(* IEC 61131-3 sources: DemoPumpStation/PumpStation/adapters/Codecs, 3 files *)

(* ---- modbus_base_codec.st ---- *)
class ModbusBaseCodec

var protected
        offset : udint := 0;
        segment : Modbus.IModbusSegmentAccess;
end_var

method public getCurrentOffset : udint
	getCurrentOffset := offset;
end_method

method protected clampInt16 : int
var_input
    value : dint;
end_var
    if value > 32767 then
        clampInt16 := 32767;
    elseif value < -32768 then
        clampInt16 := -32768;
    else
        clampInt16 := dint_to_int(value);
    end_if
end_method

method protected roundToDint : dint
var_input
    value : real;
end_var
    if value >= 0.0 then
        roundToDint := real_to_dint(value + 0.5);
    else
        roundToDint := real_to_dint(value - 0.5);
    end_if
end_method

method protected realToModbusRounded : word
var_input
	in : real;
end_var
	realToModbusRounded := int_to_word(
    						this.clampInt16(
    								this.roundToDint(in)));
end_method

method protected wordToRealValue : real
var_input in : word; end_var
	wordToRealValue := word_to_real(in);
end_method

method public init
var_input
	new_offset : uint;
	target_segment : Modbus.IModbusSegmentAccess;
end_var
offset := new_offset;
segment := target_segment;
end_method

end_class

(* ---- pdi_codec.st ---- *)
class PdiCodec extends ModbusBaseCodec

method public decode
var_in_out
    entry : PumpStationControl;
end_var
var
    cur : Modbus.ModbusCursor;
    control: word;
end_var

	if segment = NULL then return; end_if

    cur.attach(segment);
	cur.seek(offset);

	control := cur.readWord();

	entry.startCmd := control.0;
	entry.stopCmd := control.1;
	entry.setpointPower := this.wordToRealValue(cur.readWord());

    offset := cur.position();
end_method

end_class

(* ---- pdo_codec.st ---- *)
class PdoCodec extends ModbusBaseCodec

method public encode
var_input
    entry : ref_to PumpUnitView;
end_var
var
    cur : Modbus.ModbusCursor;
    states: word;
end_var

	if segment = NULL then return; end_if

    cur.attach(segment);
	cur.seek(offset);

    cur.writeDword(entry^.id);
    cur.writeWord(entry^.role);

    states.0 := entry^.available;
    states.1 := entry^.faulted;
    states.2 := entry^.active;
    cur.writeWord(states);

    cur.writeWord(this.realToModbusRounded(entry^.power));
    offset := cur.position();
end_method

method public encode
var_input
    entry : ref_to PumpControllerViewModel;
end_var
var
    cur : Modbus.ModbusCursor;
    states: word;
end_var

	if segment = NULL then return; end_if

    cur.attach(segment);
	cur.seek(offset);

	states.0 := entry^.isStarted;
	states.%b1 := entry^.vfdStatus;
	cur.writeWord(states);
	cur.writeWord(udint_to_word(entry^.vfdUnitId));
	cur.writeWord(this.realToModbusRounded(entry^.requestedPower));
	cur.writeWord(this.realToModbusRounded(entry^.vfdFrequency));
	cur.writeWord(this.realToModbusRounded(entry^.activePower));

    offset := cur.position();
end_method

end_class
